RoboDK station: Stringer C Corner-Bot-Long-BOX1.rdk

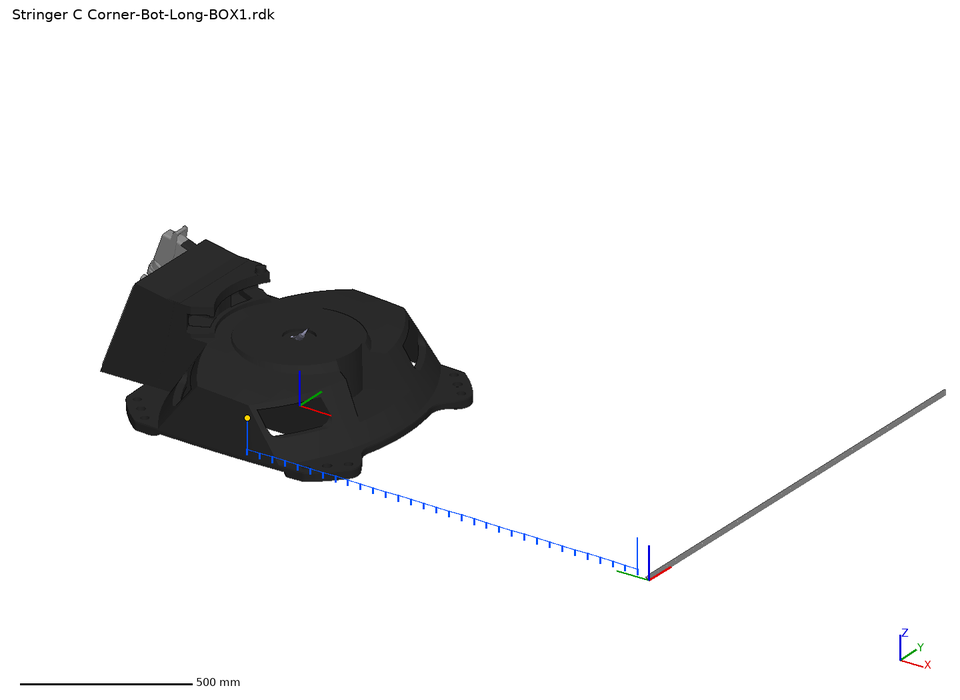
[picture v0: the station drawn from its stored meshes, robots at their saved joint values, targets as dots, program paths as lines]
Station Stringer C Corner-Bot-Long-BOX1 (saved by RoboDK 5.2.3). Poses are relative to the parent item; angles as X-Y-Z fixed-axis rotations.
  - frame KUKA KR 210 R2700 extra Base at (0, 0, 0) mm
    - robot KUKA KR 210 R2700 extra: 6 axes, payload 210 kg, reach 2696 mm, repeatability 0.06 mm, weight 1068 kg
        joint limits [-185, -140, -120, -350, -125, -350] to [185, -5, 155, 350, 125, 350]; home [0, -90, 90, 0, 0, 0]; saved at [-33.763, -51.241, 112.82, 104.469, 21.175, -132.921]
      - tool Spindle, TCP at (32, 0, 260) mm, rotated rx 0 ry 39 rz 0 deg, size 157.3 x 72 x 259.9 mm
  - frame Frame 2 at (1618.38, -541.41, 103.58) mm, rotated rx 0 ry 0 rz 90 deg
    - object Stringer C-Corner-Bot-Long-BOX1 at (0, 22.5, 0) mm, rotated rx 0 ry 0 rz -90 deg, 32 curves, geometry from Point 32
    - object L-Stringer C-Bot-Corner-Long-BOX1 at (0, 0, 0) mm, size 1499.5 x 20 x 20 mm, geometry from L-Stringer C-Bot-Corner-Long-BOX1.stl
  - machining project Point settings: rotZ(0) | rotX(0)*rotY(0) | rotz(0) | onStart | onPathStart | onApproach | onPoint | onRetract | onFinish | SetRPM(%1) | SetTool(%1) | Extruder(%1) | default | default | OutOnMov(%1) | OutOffMov(%1) | onPathFinish | M_RunCode(%1)
  - program Point (171 instructions, listed below)
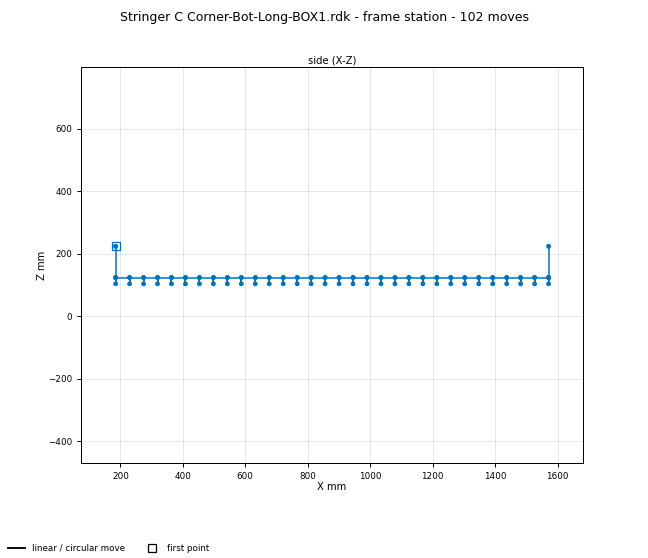
[picture p0: tool path of Stringer C Corner-Bot-Long-BOX1.rdk in frame station, 102 of 102 moves have a stored position in this frame; points joined in program order, loops and branches not executed]

--- program Point (robot KUKA KR 210 R2700 extra) ---
  Smooth(1)
  Set speed (1000.0 mm/s)
  Set Ref.: Frame 2
  Set Tool: Spindle
  Show Spindle
  MoveJ 1 to (12.5, 1433.43, 120) mm, rotated rx 180 ry 0 rz 180 deg; joints [-33.763, -56.828, 113.459, 91.551, 20.48, -119.109]
  MoveL 2 to (12.5, 1433.43, 120) mm, rotated rx 180 ry 0 rz 180 deg; joints [-33.763, -56.828, 113.459, 91.551, 20.48, -119.109]
  MoveL 3 to (12.5, 1433.43, 20) mm, rotated rx -180 ry 0 rz -180 deg; joints [-33.763, -52.025, 112.945, 102.807, 21.019, -131.14]
  MoveL 4 to (12.5, 1433.43, 20) mm, rotated rx -180 ry 0 rz -180 deg; joints [-33.763, -52.025, 112.945, 102.807, 21.019, -131.14]
  Set speed (50.0 mm/s)
  MoveL 5 to (12.5, 1433.43, 0) mm, rotated rx 180 ry 0 rz -180 deg; joints [-33.763, -51.044, 112.788, 104.877, 21.216, -133.359]
  MoveL 6 to (12.5, 1433.43, 20) mm, rotated rx -180 ry 0 rz -180 deg; joints [-33.763, -52.025, 112.945, 102.807, 21.019, -131.14]
  Set speed (1000.0 mm/s)
  MoveL 7 to (12.5, 1388.72, 20) mm, rotated rx -180 ry 0 rz -180 deg; joints [-32.416, -52.632, 114.341, 106.429, 20.592, -133.75]
  Set speed (50.0 mm/s)
  MoveL 8 to (12.5, 1388.72, 0) mm, rotated rx 180 ry 0 rz 180 deg; joints [-32.416, -51.633, 114.182, 108.547, 20.845, -136.015]
  MoveL 9 to (12.5, 1388.72, 20) mm, rotated rx -180 ry 0 rz -180 deg; joints [-32.416, -52.632, 114.341, 106.429, 20.592, -133.75]
  Set speed (1000.0 mm/s)
  MoveL 10 to (12.5, 1344.01, 20) mm, rotated rx -180 ry 0 rz -180 deg; joints [-31.027, -53.207, 115.675, 110.143, 20.213, -136.403]
  Set speed (50.0 mm/s)
  MoveL 11 to (12.5, 1344.01, 0) mm, rotated rx -180 ry 0 rz -180 deg; joints [-31.027, -52.189, 115.514, 112.293, 20.523, -138.696]
  MoveL 12 to (12.5, 1344.01, 20) mm, rotated rx -180 ry 0 rz -180 deg; joints [-31.027, -53.207, 115.675, 110.143, 20.213, -136.403]
  Set speed (1000.0 mm/s)
  MoveL 13 to (12.5, 1299.3, 20) mm, rotated rx -180 ry 0 rz -180 deg; joints [-29.596, -53.751, 116.946, 113.936, 19.88, -139.085]
  Set speed (50.0 mm/s)
  MoveL 14 to (12.5, 1299.3, 0) mm, rotated rx -180 ry 0 rz -180 deg; joints [-29.596, -52.715, 116.783, 116.101, 20.249, -141.39]
  MoveL 15 to (12.5, 1299.3, 20) mm, rotated rx -180 ry 0 rz -180 deg; joints [-29.596, -53.751, 116.946, 113.936, 19.88, -139.085]
  Set speed (1000.0 mm/s)
  MoveL 16 to (12.5, 1254.59, 20) mm, rotated rx 180 ry 0 rz 180 deg; joints [-28.124, -54.263, 118.154, 117.796, 19.593, -141.786]
  Set speed (50.0 mm/s)
  MoveL 17 to (12.5, 1254.59, 0) mm, rotated rx -180 ry 0 rz -180 deg; joints [-28.124, -53.209, 117.989, 119.957, 20.023, -144.083]
  MoveL 18 to (12.5, 1254.59, 20) mm, rotated rx 180 ry 0 rz 180 deg; joints [-28.124, -54.263, 118.154, 117.796, 19.593, -141.786]
  Set speed (1000.0 mm/s)
  MoveL 19 to (12.5, 1209.88, 20) mm, rotated rx -180 ry 0 rz -180 deg; joints [-26.61, -54.744, 119.297, 121.71, 19.35, -144.491]
  Set speed (50.0 mm/s)
  MoveL 20 to (12.5, 1209.88, 0) mm, rotated rx 180 ry 0 rz -180 deg; joints [-26.61, -53.672, 119.13, 123.847, 19.84, -146.759]
  MoveL 21 to (12.5, 1209.88, 20) mm, rotated rx -180 ry 0 rz -180 deg; joints [-26.61, -54.744, 119.297, 121.71, 19.35, -144.491]
  Set speed (1000.0 mm/s)
  MoveL 22 to (12.5, 1165.17, 20) mm, rotated rx 180 ry 0 rz 180 deg; joints [-25.055, -55.193, 120.375, 125.663, 19.149, -147.187]
  Set speed (50.0 mm/s)
  MoveL 23 to (12.5, 1165.17, 0) mm, rotated rx -180 ry 0 rz -180 deg; joints [-25.055, -54.104, 120.206, 127.756, 19.699, -149.406]
  MoveL 24 to (12.5, 1165.17, 20) mm, rotated rx 180 ry 0 rz 180 deg; joints [-25.055, -55.193, 120.375, 125.663, 19.149, -147.187]
  Set speed (1000.0 mm/s)
  MoveL 25 to (12.5, 1120.46, 20) mm, rotated rx 180 ry 0 rz -180 deg; joints [-23.459, -55.611, 121.385, 129.642, 18.986, -149.861]
  Set speed (50.0 mm/s)
  MoveL 26 to (12.5, 1120.46, 0) mm, rotated rx -180 ry 0 rz -180 deg; joints [-23.459, -54.505, 121.214, 131.67, 19.596, -152.01]
  MoveL 27 to (12.5, 1120.46, 20) mm, rotated rx 180 ry 0 rz -180 deg; joints [-23.459, -55.611, 121.385, 129.642, 18.986, -149.861]
  Set speed (1000.0 mm/s)
  MoveL 28 to (12.5, 1075.75, 20) mm, rotated rx -180 ry 0 rz -180 deg; joints [-21.824, -55.998, 122.327, 133.634, 18.859, -152.501]
  Set speed (50.0 mm/s)
  MoveL 29 to (12.5, 1075.75, 0) mm, rotated rx 180 ry 0 rz -180 deg; joints [-21.824, -54.875, 122.155, 135.578, 19.527, -154.559]
  MoveL 30 to (12.5, 1075.75, 20) mm, rotated rx -180 ry 0 rz -180 deg; joints [-21.824, -55.998, 122.327, 133.634, 18.859, -152.501]
  Set speed (1000.0 mm/s)
  MoveL 31 to (12.5, 1031.04, 20) mm, rotated rx 180 ry 0 rz 180 deg; joints [-20.151, -56.353, 123.2, 137.628, 18.764, -155.098]
  Set speed (50.0 mm/s)
  MoveL 32 to (12.5, 1031.04, 0) mm, rotated rx 180 ry 0 rz -180 deg; joints [-20.151, -55.214, 123.025, 139.469, 19.487, -157.046]
  MoveL 33 to (12.5, 1031.04, 20) mm, rotated rx 180 ry 0 rz 180 deg; joints [-20.151, -56.353, 123.2, 137.628, 18.764, -155.098]
  Set speed (1000.0 mm/s)
  MoveL 34 to (12.5, 986.33, 20) mm, rotated rx 180 ry 0 rz 180 deg; joints [-18.44, -56.677, 124.002, 141.612, 18.697, -157.642]
  Set speed (50.0 mm/s)
  MoveL 35 to (12.5, 986.33, 0) mm, rotated rx -180 ry 0 rz -180 deg; joints [-18.44, -55.523, 123.825, 143.334, 19.473, -159.463]
  MoveL 36 to (12.5, 986.33, 20) mm, rotated rx 180 ry 0 rz 180 deg; joints [-18.44, -56.677, 124.002, 141.612, 18.697, -157.642]
  Set speed (1000.0 mm/s)
  MoveL 37 to (12.5, 941.62, 20) mm, rotated rx 180 ry 0 rz -180 deg; joints [-16.696, -56.969, 124.731, 145.58, 18.654, -160.128]
  Set speed (50.0 mm/s)
  MoveL 38 to (12.5, 941.62, 0) mm, rotated rx 180 ry 0 rz 180 deg; joints [-16.696, -55.801, 124.554, 147.166, 19.478, -161.806]
  MoveL 39 to (12.5, 941.62, 20) mm, rotated rx 180 ry 0 rz -180 deg; joints [-16.696, -56.969, 124.731, 145.58, 18.654, -160.128]
  Set speed (1000.0 mm/s)
  MoveL 40 to (12.5, 896.91, 20) mm, rotated rx 180 ry 0 rz 180 deg; joints [-14.918, -57.23, 125.388, 149.525, 18.63, -162.552]
  Set speed (50.0 mm/s)
  MoveL 41 to (12.5, 896.91, 0) mm, rotated rx 180 ry 0 rz 180 deg; joints [-14.918, -56.049, 125.208, 150.963, 19.499, -164.074]
  MoveL 42 to (12.5, 896.91, 20) mm, rotated rx 180 ry 0 rz 180 deg; joints [-14.918, -57.23, 125.388, 149.525, 18.63, -162.552]
  Set speed (1000.0 mm/s)
  MoveL 43 to (12.5, 852.2, 20) mm, rotated rx 180 ry 0 rz 180 deg; joints [-13.111, -57.46, 125.97, 153.442, 18.62, -164.914]
  Set speed (50.0 mm/s)
  MoveL 44 to (12.5, 852.2, 0) mm, rotated rx 180 ry 0 rz 180 deg; joints [-13.111, -56.267, 125.789, 154.721, 19.531, -166.268]
  MoveL 45 to (12.5, 852.2, 20) mm, rotated rx 180 ry 0 rz 180 deg; joints [-13.111, -57.46, 125.97, 153.442, 18.62, -164.914]
  Set speed (1000.0 mm/s)
  MoveL 46 to (12.5, 807.49, 20) mm, rotated rx 180 ry 0 rz -180 deg; joints [-11.277, -57.658, 126.476, 157.331, 18.622, -167.215]
  Set speed (50.0 mm/s)
  MoveL 47 to (12.5, 807.49, 0) mm, rotated rx 180 ry 0 rz 180 deg; joints [-11.277, -56.455, 126.294, 158.442, 19.568, -168.39]
  MoveL 48 to (12.5, 807.49, 20) mm, rotated rx 180 ry 0 rz -180 deg; joints [-11.277, -57.658, 126.476, 157.331, 18.622, -167.215]
  Set speed (1000.0 mm/s)
  MoveL 49 to (12.5, 762.78, 20) mm, rotated rx 180 ry 0 rz -180 deg; joints [-9.42, -57.826, 126.906, 161.192, 18.631, -169.46]
  Set speed (50.0 mm/s)
  MoveL 50 to (12.5, 762.78, 0) mm, rotated rx -180 ry 0 rz -180 deg; joints [-9.42, -56.614, 126.722, 162.126, 19.608, -170.448]
  MoveL 51 to (12.5, 762.78, 20) mm, rotated rx 180 ry 0 rz -180 deg; joints [-9.42, -57.826, 126.906, 161.192, 18.631, -169.46]
  Set speed (1000.0 mm/s)
  MoveL 52 to (12.5, 718.07, 20) mm, rotated rx 180 ry 0 rz 180 deg; joints [-7.542, -57.963, 127.258, 165.026, 18.643, -171.653]
  Set speed (50.0 mm/s)
  MoveL 53 to (12.5, 718.07, 0) mm, rotated rx 180 ry 0 rz 180 deg; joints [-7.542, -56.743, 127.073, 165.778, 19.645, -172.449]
  MoveL 54 to (12.5, 718.07, 20) mm, rotated rx 180 ry 0 rz 180 deg; joints [-7.542, -57.963, 127.258, 165.026, 18.643, -171.653]
  Set speed (1000.0 mm/s)
  MoveL 55 to (12.5, 673.36, 20) mm, rotated rx 180 ry 0 rz 180 deg; joints [-5.647, -58.069, 127.531, 168.837, 18.656, -173.804]
  Set speed (50.0 mm/s)
  MoveL 56 to (12.5, 673.36, 0) mm, rotated rx -180 ry 0 rz -180 deg; joints [-5.647, -56.843, 127.346, 169.402, 19.678, -174.403]
  MoveL 57 to (12.5, 673.36, 20) mm, rotated rx 180 ry 0 rz 180 deg; joints [-5.647, -58.069, 127.531, 168.837, 18.656, -173.804]
  Set speed (1000.0 mm/s)
  MoveL 58 to (12.5, 628.65, 20) mm, rotated rx 180 ry 0 rz -180 deg; joints [-3.741, -58.144, 127.726, 172.63, 18.666, -175.922]
  Set speed (50.0 mm/s)
  MoveL 59 to (12.5, 628.65, 0) mm, rotated rx 180 ry 0 rz 180 deg; joints [-3.741, -56.913, 127.541, 173.005, 19.703, -176.32]
  MoveL 60 to (12.5, 628.65, 20) mm, rotated rx 180 ry 0 rz -180 deg; joints [-3.741, -58.144, 127.726, 172.63, 18.666, -175.922]
  Set speed (1000.0 mm/s)
  MoveL 61 to (12.5, 583.94, 20) mm, rotated rx 180 ry 0 rz 180 deg; joints [-1.825, -58.188, 127.842, 176.41, 18.673, -178.018]
  Set speed (50.0 mm/s)
  MoveL 62 to (12.5, 583.94, 0) mm, rotated rx 180 ry 0 rz -180 deg; joints [-1.825, -56.955, 127.656, 176.594, 19.719, -178.212]
  MoveL 63 to (12.5, 583.94, 20) mm, rotated rx 180 ry 0 rz 180 deg; joints [-1.825, -58.188, 127.842, 176.41, 18.673, -178.018]
  Set speed (1000.0 mm/s)
  MoveL 64 to (12.5, 539.23, 20) mm, rotated rx 180 ry 0 rz 180 deg; joints [0.094, -58.202, 127.878, 180.184, 18.676, -180.102]
  Set speed (50.0 mm/s)
  MoveL 65 to (12.5, 539.23, 0) mm, rotated rx 180 ry 0 rz 180 deg; joints [0.094, -56.968, 127.692, 180.175, 19.723, -180.092]
  MoveL 66 to (12.5, 539.23, 20) mm, rotated rx 180 ry 0 rz 180 deg; joints [0.094, -58.202, 127.878, 180.184, 18.676, -180.102]
  Set speed (1000.0 mm/s)
  MoveL 67 to (12.5, 494.52, 20) mm, rotated rx -180 ry 0 rz -180 deg; joints [2.013, -58.185, 127.834, 183.959, 18.673, -182.187]
  Set speed (50.0 mm/s)
  MoveL 68 to (12.5, 494.52, 0) mm, rotated rx -180 ry 0 rz -180 deg; joints [2.013, -56.953, 127.648, 183.756, 19.717, -181.972]
  MoveL 69 to (12.5, 494.52, 20) mm, rotated rx -180 ry 0 rz -180 deg; joints [2.013, -58.185, 127.834, 183.959, 18.673, -182.187]
  Set speed (1000.0 mm/s)
  MoveL 70 to (12.5, 449.81, 20) mm, rotated rx 180 ry 0 rz 180 deg; joints [3.927, -58.138, 127.711, 187.74, 18.665, -184.284]
  Set speed (50.0 mm/s)
  MoveL 71 to (12.5, 449.81, 0) mm, rotated rx 180 ry 0 rz 180 deg; joints [3.927, -56.908, 127.525, 187.346, 19.701, -183.866]
  MoveL 72 to (12.5, 449.81, 20) mm, rotated rx 180 ry 0 rz 180 deg; joints [3.927, -58.138, 127.711, 187.74, 18.665, -184.284]
  Set speed (1000.0 mm/s)
  MoveL 73 to (12.5, 405.11, 20) mm, rotated rx -180 ry 0 rz -180 deg; joints [5.833, -58.06, 127.508, 191.534, 18.654, -186.404]
  Set speed (50.0 mm/s)
  MoveL 74 to (12.5, 405.11, 0) mm, rotated rx 180 ry 0 rz 180 deg; joints [5.833, -56.834, 127.323, 190.95, 19.675, -185.786]
  MoveL 75 to (12.5, 405.11, 20) mm, rotated rx -180 ry 0 rz -180 deg; joints [5.833, -58.06, 127.508, 191.534, 18.654, -186.404]
  Set speed (1000.0 mm/s)
  MoveL 76 to (12.5, 360.4, 20) mm, rotated rx 180 ry 0 rz 180 deg; joints [7.726, -57.951, 127.227, 195.347, 18.642, -188.559]
  Set speed (50.0 mm/s)
  MoveL 77 to (12.5, 360.4, 0) mm, rotated rx -180 ry 0 rz -180 deg; joints [7.726, -56.731, 127.043, 194.577, 19.642, -187.743]
  MoveL 78 to (12.5, 360.4, 20) mm, rotated rx 180 ry 0 rz 180 deg; joints [7.726, -57.951, 127.227, 195.347, 18.642, -188.559]
  Set speed (1000.0 mm/s)
  MoveL 79 to (12.5, 315.69, 20) mm, rotated rx -180 ry 0 rz -180 deg; joints [9.602, -57.811, 126.867, 199.183, 18.63, -190.757]
  Set speed (50.0 mm/s)
  MoveL 80 to (12.5, 315.69, 0) mm, rotated rx -180 ry 0 rz -180 deg; joints [9.602, -56.599, 126.684, 198.232, 19.604, -189.75]
  MoveL 81 to (12.5, 315.69, 20) mm, rotated rx -180 ry 0 rz -180 deg; joints [9.602, -57.811, 126.867, 199.183, 18.63, -190.757]
  Set speed (1000.0 mm/s)
  MoveL 82 to (12.5, 270.98, 20) mm, rotated rx -180 ry 0 rz -180 deg; joints [11.457, -57.64, 126.43, 203.047, 18.622, -193.006]
  Set speed (50.0 mm/s)
  MoveL 83 to (12.5, 270.98, 0) mm, rotated rx -180 ry 0 rz -180 deg; joints [11.457, -56.438, 126.248, 201.919, 19.564, -191.814]
  MoveL 84 to (12.5, 270.98, 20) mm, rotated rx -180 ry 0 rz -180 deg; joints [11.457, -57.64, 126.43, 203.047, 18.622, -193.006]
  Set speed (1000.0 mm/s)
  MoveL 85 to (12.5, 226.27, 20) mm, rotated rx -180 ry 0 rz -180 deg; joints [13.289, -57.439, 125.916, 206.939, 18.621, -195.313]
  Set speed (50.0 mm/s)
  MoveL 86 to (12.5, 226.27, 0) mm, rotated rx 180 ry 0 rz 180 deg; joints [13.289, -56.247, 125.736, 205.643, 19.527, -193.943]
  MoveL 87 to (12.5, 226.27, 20) mm, rotated rx -180 ry 0 rz -180 deg; joints [13.289, -57.439, 125.916, 206.939, 18.621, -195.313]
  Set speed (1000.0 mm/s)
  MoveL 88 to (12.5, 181.56, 20) mm, rotated rx 180 ry 0 rz -180 deg; joints [15.093, -57.206, 125.327, 210.859, 18.631, -197.681]
  Set speed (50.0 mm/s)
  MoveL 89 to (12.5, 181.56, 0) mm, rotated rx -180 ry 0 rz -180 deg; joints [15.093, -56.026, 125.148, 209.406, 19.497, -196.144]
  MoveL 90 to (12.5, 181.56, 20) mm, rotated rx 180 ry 0 rz -180 deg; joints [15.093, -57.206, 125.327, 210.859, 18.631, -197.681]
  Set speed (1000.0 mm/s)
  MoveL 91 to (12.5, 136.85, 20) mm, rotated rx 180 ry 0 rz -180 deg; joints [16.867, -56.942, 124.664, 214.806, 18.657, -200.112]
  Set speed (50.0 mm/s)
  MoveL 92 to (12.5, 136.85, 0) mm, rotated rx 180 ry 0 rz -180 deg; joints [16.867, -55.775, 124.486, 213.206, 19.477, -198.419]
  MoveL 93 to (12.5, 136.85, 20) mm, rotated rx 180 ry 0 rz -180 deg; joints [16.867, -56.942, 124.664, 214.806, 18.657, -200.112]
  Set speed (1000.0 mm/s)
  MoveL 94 to (12.5, 92.14, 20) mm, rotated rx 180 ry 0 rz 180 deg; joints [18.609, -56.646, 123.927, 218.775, 18.703, -202.604]
  Set speed (50.0 mm/s)
  MoveL 95 to (12.5, 92.14, 0) mm, rotated rx 180 ry 0 rz 180 deg; joints [18.609, -55.494, 123.751, 217.042, 19.473, -200.769]
  MoveL 96 to (12.5, 92.14, 20) mm, rotated rx 180 ry 0 rz 180 deg; joints [18.609, -56.646, 123.927, 218.775, 18.703, -202.604]
  Set speed (1000.0 mm/s)
  MoveL 97 to (12.5, 47.43, 20) mm, rotated rx 180 ry 0 rz -180 deg; joints [20.315, -56.32, 123.118, 222.761, 18.772, -205.153]
  Set speed (50.0 mm/s)
  MoveL 98 to (12.5, 47.43, 0) mm, rotated rx 180 ry 0 rz 180 deg; joints [20.315, -55.182, 122.944, 220.91, 19.49, -203.193]
  MoveL 99 to (12.5, 47.43, 20) mm, rotated rx 180 ry 0 rz -180 deg; joints [20.315, -56.32, 123.118, 222.761, 18.772, -205.153]
  MoveL 100 to (12.5, 47.43, 20) mm, rotated rx 180 ry 0 rz -180 deg; joints [20.315, -56.32, 123.118, 222.761, 18.772, -205.153]
  Set speed (1000.0 mm/s)
  MoveL 101 to (12.5, 47.43, 20) mm, rotated rx 180 ry 0 rz -180 deg; joints [20.315, -56.32, 123.118, 222.761, 18.772, -205.153]
  MoveL 102 to (12.5, 47.43, 120) mm, rotated rx 180 ry 0 rz 180 deg; joints [20.315, -61.914, 123.688, 235.093, 15.452, -218.046]
